FUNCTION derivcvar_M_blinker_timer: LREAL
VAR_INPUT
    state: STATE;
END_VAR

derivcvar_M_blinker_timer := 1.0;

END_FUNCTION

(* stored: ProductVersion 3.1.0.18, Version 1.1.0.1 *)
